// TIA Portal V18 export
TYPE "UDT_AHsDO"
// stored: IsFailsafeCompliant false
   STRUCT
      xAHCentralEnable : Bool;
   END_STRUCT;
END_TYPE
